(* IEC 61131-3 sources: Elmo_Master/Lasal_PRG/Elmo_EtherCAT_Test_4Axis/Class/CP313_IOs, 1 file *)

(* ---- CP313_IOs.st ---- *)
(*!
<Class
	Name               = "CP313_IOs"
	Revision           = "1.1"
	RealtimeTask       = "false"
	CyclicTask         = "false"
	BackgroundTask     = "false"
	Sigmatek           = "true"
	OSInterface        = "false"
	HighPriority       = "false"
	Automatic          = "false"
	UpdateMode         = "Prescan"
	IconPath           = ".\Class\DigInOut.ICO"
	SharedCommandTable = "true"
	Objectsize         = "(622,120)"
	Comment            = "Hardwareclass to access the IOs on the CP313.">
	<Channels>
	</Channels>
	<RevDoku>
		<Owner Company="Sigmatek" Author="EisMic"/>
		<Dokumentation Revision="1.1" Date="2026-04-16" Author="LanSte" Company="Sigmatek" Description="Changed object channel To_HwControl to not required command channel."/>
		<Dokumentation Revision="1.0" Date="07.02.2020" Author="EisMic" Company="Sigmatek" Description="First library version."/>
	</RevDoku>
	<Network Name="CP313_IOs">
		<!-- List of Components in this network -->
		<Components>
			<Object
				Name       = "_base"
				Class      = "XXXBase_IOs"
				Position   = "(218,120)"
				Visualized = "false">
				<Channels>
					<Server Name="CAN_1_Connect"/>
					<Server Name="CAN_2_Connect"/>
					<Server Name="ClassState"/>
					<Server Name="COM_1_Connect"/>
					<Server Name="COM_2_Connect"/>
					<Server Name="COM_3_Connect"/>
					<Server Name="Ethernet_1_Connect"/>
					<Server Name="Ethernet_2_Connect"/>
					<Server Name="Ethernet_3_Connect"/>
					<Server Name="Ethernet_4_Connect"/>
					<Server Name="USB_1_Connect"/>
					<Client Name="To_HwControl"/>
				</Channels>
			</Object>
		</Components>
		<Comments>
		</Comments>
		<!-- List of Connections in this network -->
		<Connections>
			<Connection Source="this.ClassState" Destination="_base.ClassState" Vertices="(976,210),(804,210),"/>
			<Connection Source="this.USB_1_Connect" Destination="_base.USB_1_Connect" Vertices="(976,270),(804,270),"/>
			<Connection Source="this.CAN_1_Connect" Destination="_base.CAN_1_Connect" Vertices="(976,390),(804,570),"/>
			<Connection Source="_base.To_HwControl" Destination="this.To_HwControl" Vertices="(218,210),(38,210),"/>
			<Connection Source="this.Ethernet_1_Connect" Destination="_base.Ethernet_1_Connect" Vertices="(976,330),(804,330),"/>
		</Connections>
		<!-- Headerfiles -->
		<Options>
		</Options>
	</Network>
</Class>
*)
#pragma using XXXBase_IOs

CP313_IOs : CLASS
: XXXBase_IOs
  //Servers:
  //Clients:
  //Variables:
  //Functions:
  //Tables:
	FUNCTION @STD
		VAR_OUTPUT
			ret_code	: CONFSTATES;
		END_VAR;
	FUNCTION GLOBAL TAB @CT_;
END_CLASS;
